(* IEC 61131-3 sources: Industry-PLC-LLM/data/PLCBEAD_repo/PLCBEAD_PLCEmbed-main/PLC-BEAD/Source/GEB/HOUR_OF_DT, 1 file *)

(* ---- HOUR_OF_DT.ST ---- *)
FUNCTION HOUR_OF_DT:INT
	VAR_INPUT
		XDT :	UDINT;
	END_VAR

	HOUR_OF_DT := UDINT_TO_INT((XDT MOD UDINT#86400) / UDINT#3600);
END_FUNCTION

PROGRAM program0
  VAR
    LocalVar0 : UDINT;
	LocalOUT  : INT;
  END_VAR
  	LocalOUT := HOUR_OF_DT(LocalVar0);
END_PROGRAM
